// TIA Portal project "Motorsteuerung" (V20)

(* hardware
DEVICE "S7-1500/ET200MP-Station_1"  S7-1500 station
   slot 0: "Profilschiene_0"  Rack  6ES7 590-1***0-0AA0
   slot 1: "PLC_1"  CPU 1513-1 PN  6ES7 513-1AM03-0AB0  V4.0
      slot 3: "CPU-Display_1"  6ES7591-1AA00-0AA0
      slot 32768: "PROFINET-Schnittstelle_1"  X1
         slot 32769: "Port_1"  X1 P1
         slot 32770: "Port_2"  X1 P2
      slot 34817: "Virtual CP interface port_1"  Virtual CP interface port  Virtual CP interface port FW V4.0
   slot 2: "DI 16x24VDC BA_1"  DI 16x24VDC BA  6ES7 521-1BH10-0AA0  V1.1
   slot 3: "DQ 16x24VDC/0.5A ST_1"  DQ 16x24VDC/0.5A ST  6ES7 522-1BH00-0AB0  V2.0
   slot 4: "AI 8xU/I/R/RTD BA_2"  AI 8xU/I/R/RTD BA  6ES7 531-7QF00-0AB0  V1.0
   slot 5: "AQ 8xU/I HS_2"  AQ 8xU/I HS  6ES7 532-5HF00-0AB0  V2.2
*)

// ===== PLC "PLC_1"  CPU 1513-1 PN =====

VAR_GLOBAL   // PLC tag table "Standard-Variablentabelle"
   "Clock_Byte" AT %MB0 : Byte;
   "Clock_10Hz" AT %M0.0 : Bool;
   "Clock_5Hz" AT %M0.1 : Bool;
   "Clock_2.5Hz" AT %M0.2 : Bool;
   "Clock_2Hz" AT %M0.3 : Bool;
   "Clock_1.25Hz" AT %M0.4 : Bool;
   "Clock_1Hz" AT %M0.5 : Bool;
   "Clock_0.625Hz" AT %M0.6 : Bool;
   "Clock_0.5Hz" AT %M0.7 : Bool;
END_VAR

VAR_GLOBAL   // PLC tag table "Eingaenge"
   "Not-Aus (S1)" AT %I0.0 : Bool;
   "Linkslauf (S3)" AT %I0.1 : Bool;
   "Stopp (S2)" AT %I0.2 : Bool;
   "Rechtslauf (S4)" AT %I0.3 : Bool;
   "Linkslauf (S6)" AT %I0.5 : Bool;
   "Stopp (S5)" AT %I0.6 : Bool;
   "Rechtslauf (S7)" AT %I0.7 : Bool;
END_VAR

VAR_GLOBAL   // PLC tag table "Ausgaenge"
   "Motorschutz (H1)" AT %Q0.0 : Bool;
   "Start (H4)" AT %Q0.1 : Bool;
   "Stopp (H3)" AT %Q0.2 : Bool;
   "Start (H5)" AT %Q0.3 : Bool;
   "Motorschutz (H2)" AT %Q0.4 : Bool;
   "Start (H7)" AT %Q0.5 : Bool;
   "Stopp (H6)" AT %Q0.6 : Bool;
   "Start (H8)" AT %Q0.7 : Bool;
   "Förderer (1M1)" AT %Q1.0 : Bool;
   "Förderer (1M2)" AT %Q1.1 : Bool;
   "Förderer (2M1)" AT %A1.2 : Bool;
   "Förderer (2M2)" AT %A1.3 : Bool;
END_VAR

DATA_BLOCK "DB_Motorsteuerung"   // DB1
{ S7_Optimized_Access := 'TRUE' }
VERSION : 0.1
   VAR
      Motoren : Struct
         Motor_1 : Struct
            Motorschutz_aktiv : Bool;
            Linkslauf : Bool;
            Rechtslauf : Bool;
         END_STRUCT;
         Motor_2 : Struct
            Motorschutz_aktiv : Bool;
            Linkslauf : Bool;
            Rechtslauf : Bool;
         END_STRUCT;
      END_STRUCT;
   END_VAR
BEGIN
END_DATA_BLOCK

FUNCTION "Anlagensteuerung" : Void   // FC1, FBD
{ S7_Optimized_Access := 'TRUE' }
VERSION : 0.1
   VAR_OUTPUT
      Motor_1_Schutz : Bool;
      Motor_2_Schutz : Bool;
   END_VAR
BEGIN

REGION Network 1
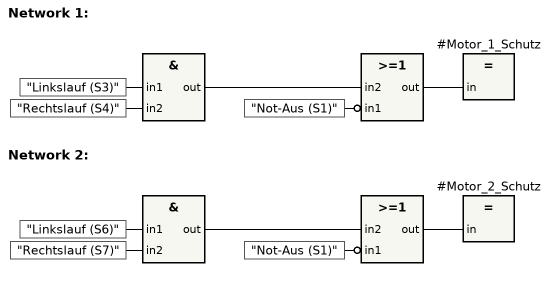
   #Motor_1_Schutz := ("Linkslauf (S3)" AND "Rechtslauf (S4)") OR NOT "Not-Aus (S1)";
END_REGION

REGION Network 2
   #Motor_2_Schutz := ("Linkslauf (S6)" AND "Rechtslauf (S7)") OR NOT "Not-Aus (S1)";
END_REGION
END_FUNCTION

FUNCTION "Foerderersteuerung" : Void   // FC2, FBD
{ S7_Optimized_Access := 'TRUE' }
VERSION : 0.1
   VAR_INPUT
      Linkslauf : Bool;
      Stopp : Bool;
      Rechtslauf : Bool;
      Motorschutz : Bool;
   END_VAR
   VAR_OUTPUT
      Motor_links : Bool;
      Motor_rechts : Bool;
   END_VAR
   VAR_IN_OUT
      Motor_links_aktiv : Bool;
      Motor_rechts_aktiv : Bool;
   END_VAR
BEGIN

REGION Network 1
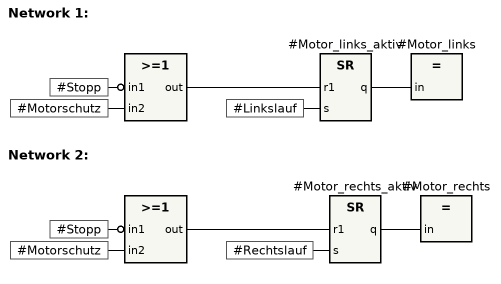
   IF #Linkslauf THEN
       #Motor_links_aktiv := TRUE;   // SR flip-flop
   END_IF;
   IF NOT #Stopp OR #Motorschutz THEN #Motor_links_aktiv := FALSE; END_IF;
   #Motor_links := #Motor_links_aktiv;
END_REGION

REGION Network 2
   IF #Rechtslauf THEN
       #Motor_rechts_aktiv := TRUE;   // SR flip-flop
   END_IF;
   IF NOT #Stopp OR #Motorschutz THEN #Motor_rechts_aktiv := FALSE; END_IF;
   #Motor_rechts := #Motor_rechts_aktiv;
END_REGION
END_FUNCTION

FUNCTION "Leuchtesteuerung" : Void   // FC3, FBD
{ S7_Optimized_Access := 'TRUE' }
VERSION : 0.1
   VAR_INPUT
      Linkslauf : Bool;
      Rechtslauf : Bool;
      Motorschutz : Bool;
      NotAus_aktiv : Bool;
   END_VAR
   VAR_OUTPUT
      Meldeleuchte_links : Bool;
      Meldeleuchte_rechts : Bool;
      Meldeleuchte_Stopp : Bool;
      Meldeleuchte_Motorschutz : Bool;
   END_VAR
BEGIN

REGION Network 1
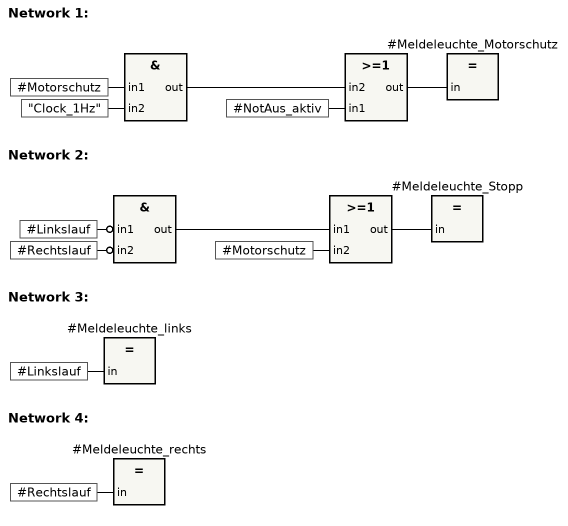
   #Meldeleuchte_Motorschutz := (#Motorschutz AND "Clock_1Hz") OR #NotAus_aktiv;
END_REGION

REGION Network 2
   #Meldeleuchte_Stopp := (NOT #Linkslauf AND NOT #Rechtslauf) OR #Motorschutz;
END_REGION

REGION Network 3
   #Meldeleuchte_links := #Linkslauf;
END_REGION

REGION Network 4
   #Meldeleuchte_rechts := #Rechtslauf;
END_REGION
END_FUNCTION

ORGANIZATION_BLOCK "Main"   // OB1, FBD, ProgramCycle
TITLE = "Main Program Sweep (Cycle)"
{ S7_Optimized_Access := 'TRUE' }
VERSION : 0.1
   VAR_INPUT
      Initial_Call : Bool;   // Initial call of this OB
      Remanence : Bool;   // =True, if remanent data are available
   END_VAR
BEGIN

REGION Network 1
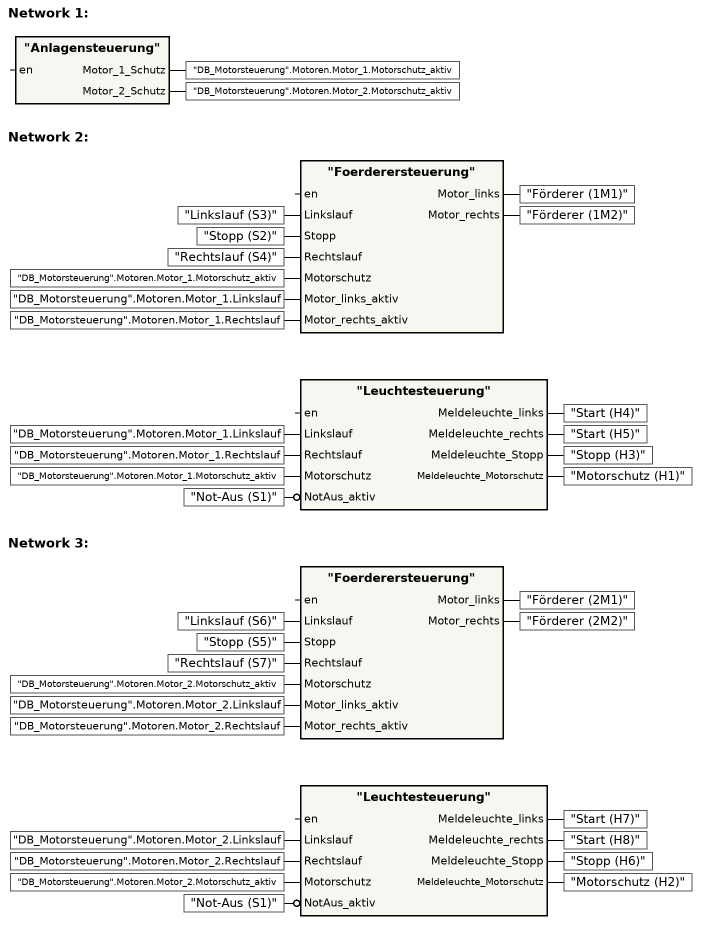
   "Anlagensteuerung"(Motor_1_Schutz => "DB_Motorsteuerung".Motoren.Motor_1.Motorschutz_aktiv,
                      Motor_2_Schutz => "DB_Motorsteuerung".Motoren.Motor_2.Motorschutz_aktiv);
END_REGION

REGION Network 2
   "Foerderersteuerung"(Linkslauf := "Linkslauf (S3)",
                        Stopp := "Stopp (S2)",
                        Rechtslauf := "Rechtslauf (S4)",
                        Motorschutz := "DB_Motorsteuerung".Motoren.Motor_1.Motorschutz_aktiv,
                        Motor_links_aktiv := "DB_Motorsteuerung".Motoren.Motor_1.Linkslauf,
                        Motor_rechts_aktiv := "DB_Motorsteuerung".Motoren.Motor_1.Rechtslauf,
                        Motor_links => "Förderer (1M1)",
                        Motor_rechts => "Förderer (1M2)");
   "Leuchtesteuerung"(Linkslauf := "DB_Motorsteuerung".Motoren.Motor_1.Linkslauf,
                      Rechtslauf := "DB_Motorsteuerung".Motoren.Motor_1.Rechtslauf,
                      Motorschutz := "DB_Motorsteuerung".Motoren.Motor_1.Motorschutz_aktiv,
                      NotAus_aktiv := NOT "Not-Aus (S1)",
                      Meldeleuchte_links => "Start (H4)",
                      Meldeleuchte_rechts => "Start (H5)",
                      Meldeleuchte_Stopp => "Stopp (H3)",
                      Meldeleuchte_Motorschutz => "Motorschutz (H1)");
END_REGION

REGION Network 3
   "Foerderersteuerung"(Linkslauf := "Linkslauf (S6)",
                        Stopp := "Stopp (S5)",
                        Rechtslauf := "Rechtslauf (S7)",
                        Motorschutz := "DB_Motorsteuerung".Motoren.Motor_2.Motorschutz_aktiv,
                        Motor_links_aktiv := "DB_Motorsteuerung".Motoren.Motor_2.Linkslauf,
                        Motor_rechts_aktiv := "DB_Motorsteuerung".Motoren.Motor_2.Rechtslauf,
                        Motor_links => "Förderer (2M1)",
                        Motor_rechts => "Förderer (2M2)");
   "Leuchtesteuerung"(Linkslauf := "DB_Motorsteuerung".Motoren.Motor_2.Linkslauf,
                      Rechtslauf := "DB_Motorsteuerung".Motoren.Motor_2.Rechtslauf,
                      Motorschutz := "DB_Motorsteuerung".Motoren.Motor_2.Motorschutz_aktiv,
                      NotAus_aktiv := NOT "Not-Aus (S1)",
                      Meldeleuchte_links => "Start (H7)",
                      Meldeleuchte_rechts => "Start (H8)",
                      Meldeleuchte_Stopp => "Stopp (H6)",
                      Meldeleuchte_Motorschutz => "Motorschutz (H2)");
END_REGION
END_ORGANIZATION_BLOCK